// TIA Portal V20 export
DATA_BLOCK "BA030AZSDR2_UnwinderBottomAxisB"   // DB263, Motion_DB
// stored: InstanceOfName TO_SynchronousAxis, OfSystemLibElement TO_SynchronousAxis, OfSystemLibVersion 9.0
TO_SynchronousAxis   // technology object, version 9.0
// stored: Connection Interface Actor, InputAddress 41232, OutputAddress 41232
// stored: Connection Interface Sensor[1], InputAddress 41232, OutputAddress 41232, SensorIndexInActorTelegram 1
// stored: Connection Interface Torque, InputAddress 64080, OutputAddress 64080
// stored: SetPointCoupling Ref BA030A_UnwinderVirtualAxis, Type TO_SynchronousAxis
   // // inherited from TO_PositioningAxis
   // // inherited from TO_SpeedAxis
   // // inherited from TO_Axis
   // // inherited from TO_Object
   // VAR
   //    Actor : TO_Struct_Actor;
   //    LoadGear : TO_Struct_LoadGear;
   //    DynamicLimits : TO_Struct_DynamicLimits;
   //    DynamicDefaults : TO_Struct_DynamicDefaults;
   // END_VAR
   // VAR
   //    Clamping : TO_Struct_Clamping;
   //    Sensor : Array[1..4] of TO_Struct_Sensor;
   //    Properties : TO_Struct_Properties;
   //    Modulo : TO_Struct_Modulo;
   //    PositionLimits_HW : TO_Struct_PositionLimitsHW;
   //    Homing : TO_Struct_Homing;
   //    PositionControl : TO_Struct_PositionControl;
   //    FollowingError : TO_Struct_FollowingError;
   //    PositioningMonitoring : TO_Struct_PositioningMonitoring;
   //    StandstillSignal : TO_Struct_StandstillSignal;
   // END_VAR
   // VAR
   //    SynchronizedMotion { S7_SetPoint := 'True'} : TO_Struct_SynchronizedMotion;
   //    StatusSynchronizedMotion { ExternalWritable := 'False'; S7_SetPoint := 'True'} : TO_Struct_StatusSynchronizedMotion;
   // END_VAR
BEGIN
   Actor.DataAdaption := 1;
   Actor.Interface.AddressIn.RID := 16#208072a;
   Actor.Interface.AddressIn.AREA := 16#81;
   Actor.Interface.AddressIn.OFFSET := 41232;
   Actor.Interface.AddressOut.RID := 16#208072b;
   Actor.Interface.AddressOut.AREA := 16#82;
   Actor.Interface.AddressOut.OFFSET := 41232;
   Actor.Interface.EnableTorqueData := true;
   Actor.Interface.TorqueDataAddressIn.RID := 16#2080742;
   Actor.Interface.TorqueDataAddressIn.AREA := 16#81;
   Actor.Interface.TorqueDataAddressIn.OFFSET := 64080;
   Actor.Interface.TorqueDataAddressOut.RID := 16#2080743;
   Actor.Interface.TorqueDataAddressOut.AREA := 16#82;
   Actor.Interface.TorqueDataAddressOut.OFFSET := 64080;
   Actor.DriveParameter.ReferenceSpeed := 8000.0;
   Actor.DriveParameter.MaxSpeed := 1300.0;
   Actor.DriveParameter.ReferenceTorque := 11.55;
   LoadGear.Numerator := 30;
   DynamicLimits.MaxVelocity := 18000.0;
   DynamicLimits.MaxAcceleration := 360000.0;
   DynamicLimits.MaxDeceleration := 360000.0;
   DynamicLimits.MaxJerk := 7200000.0;
   DynamicDefaults.Velocity := 3600.0;
   DynamicDefaults.Acceleration := 72000.0;
   DynamicDefaults.Deceleration := 72000.0;
   DynamicDefaults.Jerk := 1440000.0;
   DynamicDefaults.EmergencyDeceleration := 360000.0;
   Clamping.FollowingErrorDeviation := 360.0;
   Clamping.PositionTolerance := 360.0;
   Sensor[1]."Type" := 2;
   Sensor[1].DataAdaption := 1;
   Sensor[1].Interface.AddressIn.RID := 16#208072a;
   Sensor[1].Interface.AddressIn.AREA := 16#81;
   Sensor[1].Interface.AddressIn.OFFSET := 41232;
   Sensor[1].Interface.AddressOut.RID := 16#208072b;
   Sensor[1].Interface.AddressOut.AREA := 16#82;
   Sensor[1].Interface.AddressOut.OFFSET := 41232;
   Sensor[1].Parameter.DeterminableRevolutions := 4096;
   Properties.MotionType := 1;
   Modulo.Enable := true;
   Modulo.Length := 360.0;
   PositionLimits_HW.MinSwitchLevel := false;
   PositionLimits_HW.MaxSwitchLevel := false;
   Homing.ApproachVelocity := 3600.0;
   Homing.ReferencingVelocity := 900.0;
   PositionControl.EnableDSC := true;
   FollowingError.MinValue := 360.0;
   FollowingError.MaxValue := 3600.0;
   FollowingError.MinVelocity := 360.0;
   PositioningMonitoring.Window := 360.0;
   StandstillSignal.VelocityThreshold := 180.0;
   _Properties.MotionType := 1;
   Actor.Interface.EnableTorqueData := True;
   _Actor.Interface.Telegram := 105;
   _Actor.DataAdaptionOffline := True;
   _Sensor[1].Interface.Telegram := 105;
   _Sensor[1].DataAdaptionOffline := True;
END_DATA_BLOCK
